(* IEC 61131-3 sources: LAxisCtrl/src/blocks (part 2) *)

                            // Write MC_Command outputs to internal variable
                            _exeOfBasicMotion := 16#0;
                            _exeOfBasicMotion.%X0 := _instHalt.Busy;
                            _exeOfBasicMotion.%X1 := _instHalt.Done;
                            _exeOfBasicMotion.%X2 := _instHalt.CommandAborted;
                            _exeOfBasicMotion.%X3 := _instHalt.Error;

                        JOG_FORWARD_SELECTED, JOG_BACKWARD_SELECTED, JOG_FW_AND_BW_SELECTED:
                            // Additional features (applicative): Jog mode incremental

                            CASE _jogMode OF
                                JOG_MODE_CONTINUOUS:

                                    // No additional feature
                                    // Firstcycle of command
                                    IF (_firstCycleBasicMotion = TRUE) THEN
                                        // Copy no dynamics into static variables because changes are accepted by MC_MoveJog immediately (enable)
                                        _instMoveJog(Axis := _refSpeedAxis^,
                                                     JogForward := FALSE,
                                                     JogBackward := FALSE);
                                    END_IF;

                                    // Call MC_Command
                                    _instMoveJog(Axis := _refSpeedAxis^,
                                                 JogForward := _basicCommand.%X2,
                                                 JogBackward := _basicCommand.%X3,
                                                 Velocity := config.jog.velocity,
                                                 Acceleration := config.jog.acceleration,
                                                 Deceleration := config.jog.deceleration,
                                                 PositionControlled := config.jog.positionControlled,
                                                 Jerk := config.jog.jerk);

                                    // Evaluate MC_Command
                                    IF (_instMoveJog.Busy = FALSE) AND
                                        (_instMoveJog.Error = FALSE) AND
                                        (_instMoveJog.CommandAborted = FALSE) AND
                                        (_instMoveJog.InVelocity = FALSE)
                                    THEN
                                        // Return to NO_SELECTION if command finished
                                        _basicMotionState := NO_SELECTION;

                                    ELSIF (_instMoveJog.Error = TRUE) THEN
                                        // Errorhandling
                                        _status := AxisStatus#ERR_MC_MOVEJOG;
                                        _statusText := STRING#'ERR_MC_MOVEJOG';
                                        _errorAutoCleared := TRUE;
                                        _diagnostics.subfunctionStatus := _instMoveJog.ErrorId;
                                        _subfunctionStatus := _instMoveJog.ErrorId;
                                        // Set next state
                                        _basicMotionState := NO_SELECTION;
                                        _state := AXIS_STOP_ON_ERROR_SELECTION;
                                        // ELSE
                                        //   ; // Command selected
                                    END_IF;

                                    // Write MC_Command outputs to internal variable
                                    _exeOfBasicMotion := 16#0;
                                    _exeOfBasicMotion.%X0 := _instMoveJog.Busy;
                                    _exeOfBasicMotion.%X2 := _instMoveJog.CommandAborted;
                                    _exeOfBasicMotion.%X3 := _instMoveJog.Error;
                                    _exeOfBasicMotion.%X4 := _instMoveJog.InVelocity;

                                JOG_MODE_CONTINUE_INCREMENT, JOG_MODE_NEW_INCREMENT:

                                    // This case is additional feature (MC_MOVERELATIVE and MC_HALT internal used)
                                    CASE _exeOfBasicMotion OF
                                        CMD_BUSY:
                                            // Firstcycle of command
                                            IF (_firstCycleBasicMotion = TRUE) THEN // New rising edge at JogForward or JogBackward
                                                // Check for only one Jog direction selected (Forward OR Backward)
                                                IF (_basicCommand.%X2 XOR _basicCommand.%X3) // Only one direction selected
                                                THEN
                                                    // Reset MOVERELATIVE command
                                                    _instMoveRelative(Axis := _refPosAxis^,
                                                                      Execute := FALSE);
                                                    // Reset HALT command
                                                    _instHalt(Axis := _refSpeedAxis^,
                                                              Execute := FALSE);

                                                    // Set new Increment if direction changed necessary
                                                    IF (_resetIncJog = FALSE) THEN
                                                        IF ((_incJogDirectionOld = FORWARD_DIR) AND (_basicCommand.%X2 = TRUE)) OR
                                                            ((_incJogDirectionOld = BACKWARD_DIR) AND (_basicCommand.%X3 = TRUE))
                                                        THEN
                                                            ; // Direction of last jog process same as current --> continue Jog
                                                        ELSE
                                                            _resetIncJog := TRUE;
                                                        END_IF;
                                                    END_IF;

                                                    // Determine distance for positioning command (relative)
                                                    IF (config.jog.mode = JOG_MODE_NEW_INCREMENT) // In this mode a new increment is always set
                                                        OR ((config.jog.mode = JOG_MODE_CONTINUE_INCREMENT) AND (_resetIncJog = TRUE))
                                                    THEN
                                                        _resetIncJog := FALSE;
                                                        // New increment
                                                        IF (_refPosAxis <> NULL) THEN // Axis type is TO_PositioningAxis or TO_SynchronousAxis
                                                            _incJogStartPosition := _refPosAxis^.Position;
                                                        ELSE // Invalid TO specification
                                                            _incJogStartPosition := 0.0;
                                                        END_IF;
                                                        _increment := Abs(config.jog.increment); // absolute Distance for increment
                                                        IF (_basicCommand.%X2 = TRUE) THEN
                                                            // JogForward selected
                                                            _position := Abs(config.jog.increment);
                                                            _increment := _position;
                                                            _incJogDirectionOld := FORWARD_DIR;
                                                        ELSIF (_basicCommand.%X3 = TRUE) THEN
                                                            // JogBackward selected
                                                            _position := -Abs(config.jog.increment);
                                                            _increment := _position;
                                                            _incJogDirectionOld := BACKWARD_DIR;
                                                        ELSE
                                                            // Normal not possible to reach ELSE-branch
                                                            _incJogDirectionOld := 0;
                                                        END_IF;
                                                    ELSE
                                                        // Check for modulo axis
                                                        IF (_refPosAxis <> NULL) THEN // Axis type is TO_PositioningAxis or TO_SynchronousAxis
                                                            tempBool := _refPosAxis^.Modulo.Enable;
                                                        ELSE // Invalid TO specification
                                                            tempBool := FALSE;
                                                        END_IF;

                                                        IF (tempBool = FALSE) THEN
                                                            // No Modulo enabled
                                                            // Continue increment
                                                            IF (_refPosAxis <> NULL) THEN // Axis type is TO_PositioningAxis or TO_SynchronousAxis
                                                                tempLReal := _refPosAxis^.Position;
                                                            ELSE // Invalid TO specification
                                                                tempLReal := 0.0;
                                                            END_IF;

                                                            _position := (_incJogStartPosition + _increment) - tempLReal;
                                                            // Distance := setpoint - actualvalue
                                                        ELSE
                                                            // Modulo enabled
                                                            _position := _incJogDistance;
                                                        END_IF;
                                                    END_IF;
                                                    _incJogSubState := INC_JOG_START;

                                                    // Store Dynamics
                                                    _basicVelocity := Abs(config.jog.velocity);
                                                    _basicAcceleration := config.jog.acceleration;
                                                    _basicDeceleration := config.jog.deceleration;
                                                    _basicJerk := config.jog.jerk;
                                                ELSE
                                                    // Errorhandling - Invalid direction (forward and backward selected)
                                                    _status := AxisStatus#ERR_INVALID_JOG_DIR;
                                                    _statusText := STRING#'ERR_INVALID_JOG_DIR';
                                                    _errorAutoCleared := TRUE;
                                                    _diagnostics.subfunctionStatus := WORD#0000;
                                                    _subfunctionStatus := AxisStatus#STATUS_NO_CALL;
                                                    _diagnostics.basicMotionState := _basicMotionState;
                                                    // Set next state
                                                    _state := AXIS_STOP_ON_ERROR_SELECTION;
                                                    _basicMotionState := NO_SELECTION;
                                                    _exeOfBasicMotion := CMD_ERROR;
                                                    _incJogSubState := INC_JOG_IDLE;
                                                END_IF;

                                            ELSIF ((_basicCommand.%X2 = FALSE) AND (_basicCommand.%X3 = FALSE)) // No jog input selected --> Stop moving
                                                AND (_incJogSubState <> INC_JOG_STOP)
                                            THEN
                                                // Reset HALT command
                                                _instHalt(Axis := _refSpeedAxis^,
                                                          Execute := FALSE);
                                                _incJogSubState := INC_JOG_STOP;
                                                IF (_refPosAxis <> NULL) THEN // Axis type is TO_PositioningAxis or TO_SynchronousAxis
                                                    _incJogDistance := _refPosAxis^.StatusPositioning.Distance;
                                                ELSE // Invalid TO specification
                                                    _incJogDistance := 0.0;
                                                END_IF;

                                            ELSIF (_basicCommand.%X2 = TRUE) AND (_basicCommand.%X3 = TRUE) // jogForward and jogBackward selected - Error
                                            THEN
                                                // Reset HALT command
                                                _instHalt(Axis := _refSpeedAxis^,
                                                         Execute := FALSE);
                                                _incJogSubState := INC_JOG_STOP;
                                                // Errorhandling
                                                _status := AxisStatus#ERR_INVALID_JOG_DIR;
                                                _statusText := STRING#'ERR_INVALID_JOG_DIR';
                                                _errorAutoCleared := TRUE;
                                                _diagnostics.subfunctionStatus := WORD#0000;
                                                _subfunctionStatus := AxisStatus#STATUS_NO_CALL;
                                                // Set next state
                                                _exeOfBasicMotion := CMD_ERROR;
                                                _basicMotionState := NO_SELECTION;
                                                _state := AXIS_STOP_ON_ERROR_SELECTION;
                                            // ELSE
                                                //   ; // Command running
                                            END_IF;

                                            // Select motion
                                            CASE _incJogSubState OF
                                                INC_JOG_IDLE:
                                                    ; // Do nothing - Error occurred (jogforward and jogbackward are set in firstCycle of operation)

                                                INC_JOG_START: // Run jog operation --> Motion stops automatically if increment complete
                                                    _instMoveRelative(Axis := _refPosAxis^,
                                                                    Execute := TRUE,
                                                                    Distance := _position,
                                                                    Velocity := _basicVelocity,
                                                                    Acceleration := _basicAcceleration,
                                                                    Deceleration := _basicDeceleration,
                                                                    Jerk := _basicJerk);

                                                // Evaluate MC_Command
                                                IF (_instMoveRelative.Done = TRUE) THEN
                                                    // Increment completed
                                                    _resetIncJog := TRUE;
                                                    // Set next state
                                                    _exeOfBasicMotion := CMD_DONE;
                                                    _incJogSubState := INC_JOG_IDLE;

                                                ELSIF (_instMoveRelative.Error = TRUE) THEN
                                                    _resetIncJog := TRUE;
                                                    // Errorhandling
                                                    _status := AxisStatus#ERR_MC_MOVERELATIVE;
                                                    _statusText := STRING#'ERR_MC_MOVERELATIVE';
                                                    _errorAutoCleared := TRUE;
                                                    _diagnostics.subfunctionStatus := _instMoveRelative.ErrorId;
                                                    _subfunctionStatus := _instMoveRelative.ErrorId;
                                                    // Set next state
                                                    _state := AXIS_STOP_ON_ERROR_SELECTION;
                                                    _basicMotionState := NO_SELECTION;
                                                    _exeOfBasicMotion := CMD_ERROR;
                                                    _incJogSubState := INC_JOG_IDLE;

                                                ELSIF (_instMoveRelative.CommandAborted = TRUE) THEN
                                                    _resetIncJog := TRUE;
                                                    _exeOfBasicMotion := CMD_ABORTED;
                                                    _incJogSubState := INC_JOG_IDLE;
                                                    // ELSE
                                                    //   ; // Wait for next state
                                                END_IF;

                                                INC_JOG_STOP: // Executed if inputs are reset --> Stop jog operation OR if jogForward and jogBackward are set --> Error and stop axis
                                                    _instHalt(Axis := _refSpeedAxis^,
                                                              Execute := TRUE,
                                                              Deceleration := _basicDeceleration,
                                                              AbortAcceleration := FALSE,
                                                              Jerk := _basicJerk,
                                                              Mode := 0); // Mode := 0 "The basic motion and the superimposed motion are stopped." MC_Halt instance is also used for input 'stop', where the 'haltMode' can now be specified via config

                                                    // Evaluate MC_Command
                                                    IF (_instHalt.Done = TRUE) THEN
                                                        // Set next state
                                                        _exeOfBasicMotion := CMD_END_PROCESS;
                                                        _incJogSubState := INC_JOG_IDLE;

                                                    ELSIF (_instHalt.Error = TRUE) THEN
                                                        _resetIncJog := TRUE;
                                                        // Errorhandling
                                                        _status := AxisStatus#ERR_MC_HALT;
                                                        _statusText := STRING#'ERR_MC_HALT';
                                                        _errorAutoCleared := TRUE;
                                                        _diagnostics.subfunctionStatus := _instHalt.ErrorId;
                                                        _subfunctionStatus := _instHalt.ErrorId;
                                                        // Set next state
                                                        _state := AXIS_STOP_ON_ERROR_SELECTION;
                                                        _basicMotionState := NO_SELECTION;
                                                        _exeOfBasicMotion := CMD_ERROR;
                                                        _incJogSubState := INC_JOG_IDLE;

                                                    ELSIF (_instHalt.CommandAborted = TRUE) THEN
                                                        _resetIncJog := TRUE;
                                                        // Set next state
                                                        _incJogSubState := INC_JOG_IDLE;
                                                        _exeOfBasicMotion := CMD_ABORTED;
                                                    // ELSE
                                                        //   ; // Wait for stopping axis
                                                    END_IF;
                                                ELSE
                                                    // Errorhandling
                                                    _status := AxisStatus#ERR_UNDEFINED_INCREMENTAL_JOG_SUBSTATE;
                                                    _statusText := STRING#'ERR_UNDEFINED_INCREMENTAL_JOG_SUBSTATE';
                                                    _errorUserCleared := TRUE;
                                                    _diagnostics.subfunctionStatus := WORD#0000;
                                                    _subfunctionStatus := AxisStatus#STATUS_NO_CALL;
                                                    // Set errorstate
                                                    _state := FB_ERROR;
                                                END_CASE;

                                        CMD_DONE,
                                        CMD_ABORTED,
                                        CMD_ERROR,
                                        CMD_END_PROCESS:
                                            // Return to NO_SELECTION if command finished
                                            IF (_basicCommand.%X2 = FALSE) AND (_basicCommand.%X3 = FALSE) THEN
                                                // jogForward and jogbackward inputs are reset
                                                _exeOfBasicMotion := CMD_BUSY;
                                                _basicMotionState := NO_SELECTION;
                                            // ELSE
                                                //   ; // Wait for falling edge at inputs for jog
                                            END_IF;
                                    ELSE
                                        // Errorhandling
                                        _status := AxisStatus#ERR_UNDEFINED_INCREMENTAL_JOG_STATE;
                                        _statusText := STRING#'ERR_UNDEFINED_INCREMENTAL_JOG_STATE';
                                        _errorUserCleared := TRUE;
                                        _diagnostics.subfunctionStatus := WORD#0000;
                                        _subfunctionStatus := AxisStatus#STATUS_NO_CALL;
                                        _diagnostics.basicMotionState := _basicMotionState;
                                        // Set errorstate
                                        _state := FB_ERROR;
                                    END_CASE;

                            ELSE
                                // Errorhandling - Invalid jog state
                                _status := AxisStatus#ERR_INVALID_JOG_MODE;
                                _statusText := STRING#'#ERR_INVALID_JOG_MODE';
                                _errorAutoCleared := TRUE;
                                _diagnostics.subfunctionStatus := WORD#0000;
                                _subfunctionStatus := AxisStatus#STATUS_NO_CALL;
                                // Set next state
                                _state := AXIS_STOP_ON_ERROR_SELECTION;
                                _basicMotionState := NO_SELECTION;
                            END_CASE;

                        MOVE_VELOCITY_SELECTED:
                            // Additional features (applicative): Change setpoint on the fly (Velocity)

                            // Firstcycle of command
                            IF (_firstCycleBasicMotion = TRUE) THEN
                                // Reset MC_MOVEVELOCITY command
                                _instMoveVelocity(Axis := _refSpeedAxis^,
                                                    Execute := FALSE);

                                _velocityChangeOnTheFly := config.moveVelocity.velocityChangeOnTheFly;

                                _instMoveVelocity.Velocity := config.moveVelocity.velocity;
                                _basicVelocity := config.moveVelocity.velocity;

                                _instMoveVelocity.Acceleration := config.moveVelocity.acceleration;
                                _instMoveVelocity.Deceleration := config.moveVelocity.deceleration;
                                _instMoveVelocity.Jerk := config.moveVelocity.jerk;
                                _instMoveVelocity.Direction := config.moveVelocity.direction;
                                _instMoveVelocity.PositionControlled := config.moveVelocity.positionControlled;
                                _instMoveVelocity.Current := FALSE;

                            ELSIF (_velocityChangeOnTheFly = TRUE) AND (config.moveVelocity.velocity <> _basicVelocity) // Velocity changed
                                AND (_instMoveVelocity.CommandAborted = FALSE)
                            THEN
                                // Reset MC_MOVEVELOCITY command
                                _instMoveVelocity(Axis := _refSpeedAxis^,
                                                Execute := FALSE);

                                _instMoveVelocity.Velocity := config.moveVelocity.velocity;
                                _basicVelocity := config.moveVelocity.velocity;

                                // Copy also dynamics
                                _instMoveVelocity.Acceleration := config.moveVelocity.acceleration;
                                _instMoveVelocity.Deceleration := config.moveVelocity.deceleration;
                                _instMoveVelocity.Jerk := config.moveVelocity.jerk;
                                _instMoveVelocity.Direction := config.moveVelocity.direction;
                                _instMoveVelocity.PositionControlled := config.moveVelocity.positionControlled;
                            END_IF;

                            // Call MC_Command
                            _instMoveVelocity(Axis := _refSpeedAxis^,
                                              Execute := _basicCommand.%X4 OR _firstCycleBasicMotion); // Input: moveVelocity

                            // Evaluate MC_Command
                            IF (_instMoveVelocity.Busy = FALSE) AND
                                (_instMoveVelocity.Error = FALSE) AND
                                (_instMoveVelocity.CommandAborted = FALSE) AND
                                (_instMoveVelocity.InVelocity = FALSE)
                            THEN
                                // Return to NO_SELECTION if command finished
                                _basicMotionState := NO_SELECTION;

                            ELSIF (_instMoveVelocity.Error = TRUE) THEN
                                // Errorhandling
                                _status := AxisStatus#ERR_MC_MOVEVELOCITY;
                                _statusText := STRING#'ERR_MC_MOVEVELOCITY';
                                _errorAutoCleared := TRUE;
                                _diagnostics.subfunctionStatus := _instMoveVelocity.ErrorId;
                                _subfunctionStatus := _instMoveVelocity.ErrorId;
                                _velocityChangeOnTheFly := FALSE;
                                // Set next state
                                _state := AXIS_STOP_ON_ERROR_SELECTION;
                                _basicMotionState := NO_SELECTION;
                                // ELSE
                                //   ; // Command selected
                            END_IF;

                            // Write MC_Command outputs to internal variable
                            _exeOfBasicMotion := 16#0;
                            _exeOfBasicMotion.%X0 := _instMoveVelocity.Busy;
                            _exeOfBasicMotion.%X2 := _instMoveVelocity.CommandAborted;
                            _exeOfBasicMotion.%X3 := _instMoveVelocity.Error;
                            _exeOfBasicMotion.%X4 := _instMoveVelocity.InVelocity;

                        POS_RELATIVE_SELECTED:
                            // Additional features (applicative): Specified direction

                            // Firstcycle of command
                            IF (_firstCycleBasicMotion = TRUE) THEN
                                // Configurate the direction of rotation
                                IF ((config.posRelative.direction = 0) AND (config.posRelative.distance >= 0.0)) // Sign of distance is evaluated
                                    OR (config.posRelative.direction = FORWARD_DIR) // Forward direction
                                THEN
                                    _position := Abs(config.posRelative.distance);
                                    // Reset MC_MOVERELATIVE command
                                    _instMoveRelative(Axis := _refPosAxis^,
                                                      Execute := FALSE,
                                                      Distance := _position,
                                                      Velocity := config.posRelative.velocity,
                                                      Acceleration := config.posRelative.acceleration,
                                                      Deceleration := config.posRelative.deceleration,
                                                      Jerk := config.posRelative.jerk);
                                    _applicativeBasicMotionError := FALSE;

                                ELSIF ((config.posRelative.direction = 0) AND (config.posRelative.distance < 0.0)) // Sign of distance is evaluated
                                    OR (config.posRelative.direction = BACKWARD_DIR) // Backward direction
                                THEN
                                    _position := -Abs(config.posRelative.distance);
                                    // Reset MC_MOVERELATIVE command
                                    _instMoveRelative(Axis := _refPosAxis^,
                                                      Execute := FALSE,
                                                      Distance := _position,
                                                      Velocity := config.posRelative.velocity,
                                                      Acceleration := config.posRelative.acceleration,
                                                      Deceleration := config.posRelative.deceleration,
                                                      Jerk := config.posRelative.jerk);

                                    _applicativeBasicMotionError := FALSE;
                                ELSE
                                    // Errorhandling - Invalid direction
                                    _status := AxisStatus#ERR_INVALID_POS_RELATIVE_DIR;
                                    _statusText := STRING#'ERR_INVALID_POS_RELATIVE_DIR';
                                    _errorAutoCleared := TRUE;
                                    _diagnostics.subfunctionStatus := WORD#0000;
                                    _subfunctionStatus := AxisStatus#STATUS_NO_CALL;
                                    _applicativeBasicMotionError := TRUE;
                                    // Set next state
                                    _state := AXIS_STOP_ON_ERROR_SELECTION;
                                    _basicMotionState := NO_SELECTION;
                                END_IF;
                            END_IF;

                            IF (_applicativeBasicMotionError = FALSE) THEN
                                // Call MC_Command
                                _instMoveRelative(Axis := _refPosAxis^,
                                                  Execute := _basicCommand.%X5 OR _firstCycleBasicMotion); // Input: posRelative

                                // Evaluate MC_Command
                                IF (_instMoveRelative.Busy = FALSE) AND
                                    (_instMoveRelative.Error = FALSE) AND
                                    (_instMoveRelative.Done = FALSE) AND
                                    (_instMoveRelative.CommandAborted = FALSE)
                                THEN
                                    // Return to NO_SELECTION if command finished
                                    _basicMotionState := NO_SELECTION;

                                ELSIF (_instMoveRelative.Error = TRUE) THEN
                                    // Errorhandling
                                    _status := AxisStatus#ERR_MC_MOVERELATIVE;
                                    _statusText := STRING#'ERR_MC_MOVERELATIVE';
                                    _errorAutoCleared := TRUE;
                                    _diagnostics.subfunctionStatus := _instMoveRelative.ErrorId;
                                    _subfunctionStatus := _instMoveRelative.ErrorId;
                                    // Set next state
                                    _state := AXIS_STOP_ON_ERROR_SELECTION;
                                    _basicMotionState := NO_SELECTION;
                                // ELSE
                                    //   ; // Command selected
                                END_IF;

                                // Write MC_Command outputs to internal variable
                                _exeOfBasicMotion := 16#0;
                                _exeOfBasicMotion.%X0 := _instMoveRelative.Busy;
                                _exeOfBasicMotion.%X1 := _instMoveRelative.Done;
                                _exeOfBasicMotion.%X2 := _instMoveRelative.CommandAborted;
                                _exeOfBasicMotion.%X3 := _instMoveRelative.Error;
                            // ELSE
                                //   ; // Direction not valid
                            END_IF;

                        POS_ABSOLUTE_SELECTED:
                            // Additional features (applicative): Change setpoint on the fly (Velocity and Position)

                            // Firstcycle of command
                            IF (_firstCycleBasicMotion = TRUE) THEN
                                // Reset MC_MOVEABSOLUTE command
                                _instMoveAbsolute(Axis := _refPosAxis^,
                                                  Execute := FALSE);

                                _instMoveAbsolute.Position := config.posAbsolute.position;
                                _position := config.posAbsolute.position;
                                _instMoveAbsolute.Velocity := config.posAbsolute.velocity;
                                _basicVelocity := config.posAbsolute.velocity;

                                _instMoveAbsolute.Acceleration := config.posAbsolute.acceleration;
                                _instMoveAbsolute.Deceleration := config.posAbsolute.deceleration;
                                _instMoveAbsolute.Jerk := config.posAbsolute.jerk;
                                _instMoveAbsolute.Direction := config.posAbsolute.direction;

                                _velocityChangeOnTheFly := config.posAbsolute.velocityChangeOnTheFly;
                                _positionChangeOnTheFly := config.posAbsolute.positionChangeOnTheFly;

                            ELSIF (((_velocityChangeOnTheFly = TRUE) AND (config.posAbsolute.velocity <> _basicVelocity))
                                OR ((_positionChangeOnTheFly = TRUE) AND (config.posAbsolute.position <> _position)))
                                AND (_instMoveAbsolute.CommandAborted = FALSE)
                            THEN
                                // Reset MC_MOVEABSOLUTE command
                                _instMoveAbsolute(Axis := _refPosAxis^,
                                                  Execute := FALSE);

                                IF (_velocityChangeOnTheFly = TRUE) THEN // Apply the new velocity value
                                    _instMoveAbsolute.Velocity := config.posAbsolute.velocity;
                                    _basicVelocity := config.posAbsolute.velocity;

                                    // Copy also dynamics
                                    _instMoveAbsolute.Acceleration := config.posAbsolute.acceleration;
                                    _instMoveAbsolute.Deceleration := config.posAbsolute.deceleration;
                                    _instMoveAbsolute.Jerk := config.posAbsolute.jerk;
                                    _instMoveAbsolute.Direction := config.posAbsolute.direction;
                                END_IF;

                                IF (_positionChangeOnTheFly = TRUE) THEN // Apply the new position value
                                    _instMoveAbsolute.Position := config.posAbsolute.position;
                                    _position := config.posAbsolute.position;

                                    // Copy also dynamics
                                    _instMoveAbsolute.Velocity := config.posAbsolute.velocity;
                                    _instMoveAbsolute.Acceleration := config.posAbsolute.acceleration;
                                    _instMoveAbsolute.Deceleration := config.posAbsolute.deceleration;
                                    _instMoveAbsolute.Jerk := config.posAbsolute.jerk;
                                    _instMoveAbsolute.Direction := config.posAbsolute.direction;
                                END_IF;
                            END_IF;

                            _instMoveAbsolute(Axis := _refPosAxis^,
                                              Execute := _basicCommand.%X6 OR _firstCycleBasicMotion); // Input: posAbsolute

                            // Evaluate MC_Command
                            IF (_instMoveAbsolute.Busy = FALSE) AND
                                (_instMoveAbsolute.Error = FALSE) AND
                                (_instMoveAbsolute.Done = FALSE) AND
                                (_instMoveAbsolute.CommandAborted = FALSE)
                            THEN
                                // Return to NO_SELECTION if command finished
                                _basicMotionState := NO_SELECTION;

                            ELSIF (_instMoveAbsolute.Error = TRUE) THEN
                                // Errorhandling
                                _status := AxisStatus#ERR_MC_MOVEABSOLUTE;
                                _statusText := STRING#'ERR_MC_MOVEABSOLUTE';
                                _errorAutoCleared := TRUE;
                                _diagnostics.subfunctionStatus := _instMoveAbsolute.ErrorId;
                                _subfunctionStatus := _instMoveAbsolute.ErrorId;
                                _velocityChangeOnTheFly := FALSE;
                                _positionChangeOnTheFly := FALSE;
                                // Set next state
                                _state := AXIS_STOP_ON_ERROR_SELECTION;
                                _basicMotionState := NO_SELECTION;
                            END_IF;

                            // Write MC_Command outputs to internal variable
                            _exeOfBasicMotion := 16#0;
                            _exeOfBasicMotion.%X0 := _instMoveAbsolute.Busy;
                            _exeOfBasicMotion.%X1 := _instMoveAbsolute.Done;
                            _exeOfBasicMotion.%X2 := _instMoveAbsolute.CommandAborted;
                            _exeOfBasicMotion.%X3 := _instMoveAbsolute.Error;

                        ACTIVE_HOMING_SELECTED:
                            // Additional feature (applicative): homing on fixed stop

                            // Firstcycle of command
                            IF (_firstCycleBasicMotion = TRUE) THEN
                                _activeHomingState := config.homing.extendedMode;
                                _exeOfBasicMotion := CMD_BUSY;
                                _passiveHomingState := NO_HOMING_ACTIVE;
                            END_IF;

                            // Selection of extended homing mode
                            CASE _activeHomingState OF
                                STANDARD_HOMING:
                                    // No additional features

                                    // Firstcycle of command
                                    IF (_firstCycleBasicMotion = TRUE) THEN
                                        // Reset MC_HOME command
                                        _instHome(Axis := _refAxis^,
                                                  Execute := FALSE,
                                                  Position := config.homing.position,
                                                  Mode := config.homing.mode,
                                                  Sensor := config.homing.sensor);
                                    END_IF;

                                    // Call MC_Command

                                    _instHome(Axis := _refAxis^,
                                              Execute := _basicCommand.%X10 OR _firstCycleBasicMotion); // Input: homing

                                    // Evaluate MC_Command
                                    IF (_instHome.Busy = FALSE) AND
                                        (_instHome.Done = FALSE) AND
                                        (_instHome.CommandAborted = FALSE) AND
                                        (_instHome.Error = FALSE)
                                    THEN
                                        // Return to NO_SELECTION if command finished
                                        _activeHomingState := STANDARD_HOMING;
                                        _basicMotionState := NO_SELECTION;

                                    ELSIF (_instHome.Error = TRUE) THEN
                                        // Errorhandling
                                        _status := AxisStatus#ERR_MC_HOME;
                                        _statusText := STRING#'ERR_MC_HOME';
                                        _errorAutoCleared := TRUE;
                                        _diagnostics.subfunctionStatus := _instHome.ErrorId;
                                        _subfunctionStatus := _instHome.ErrorId;
                                        _state := AXIS_STOP_ON_ERROR_SELECTION;
                                        _basicMotionState := NO_SELECTION;
                                        // ELSE
                                        //   ; // Command selected
                                    END_IF;

                                    _exeOfBasicMotion := 16#0;
                                    _exeOfBasicMotion.%X0 := _instHome.Busy;
                                    _exeOfBasicMotion.%X1 := _instHome.Done;
                                    _exeOfBasicMotion.%X2 := _instHome.CommandAborted;
                                    _exeOfBasicMotion.%X3 := _instHome.Error;

                                HOMING_ON_FIXED_STOP,
                                HOMING_ON_FIXED_STOP_WITH_MOVING_OUT_OF_CLAMPING,
                                HOMING_ON_FIXED_STOP_WITH_MOVING_TO_TARGET_POSITION:
                                    // This case is additional feature (MC_MOVEVELOCITY and MC_HOME internal used)

                                    CASE _exeOfBasicMotion OF
                                        CMD_BUSY:
                                            // Firstcycle of command
                                            IF (_firstCycleBasicMotion = TRUE) THEN

                                                // Read operative sensor
                                                IF (_refPosAxis <> NULL) THEN // Axis type is TO_PositioningAxis or TO_SynchronousAxis
                                                    tempIndex := TO_INT(_refPosAxis^.OperativeSensor);
                                                ELSE // Invalid TO specification
                                                    tempIndex := 1;
                                                END_IF;

                                                IF (tempIndex < 1) THEN
                                                    tempIndex := 1;
                                                END_IF;

                                                IF (_refPosAxis <> NULL) THEN // Axis type is TO_PositioningAxis or TO_SynchronousAxis
                                                    tempDInt := _refPosAxis^.Sensor[tempIndex].ActiveHoming.Direction;
                                                ELSE // Invalid TO specification
                                                    tempDInt := 0; // Positive direction
                                                END_IF;

                                                IF (tempDInt = 0)
                                                THEN
                                                    // Positive direction
                                                    _direction := FORWARD_DIR;
                                                ELSE
                                                    // Negative direction
                                                    _direction := BACKWARD_DIR;
                                                END_IF;

                                                // Check if homing on fixed stop is allowed

                                                IF (_refPosAxis <> NULL) THEN // Axis type is TO_PositioningAxis or TO_SynchronousAxis
                                                    tempBool := _refPosAxis^.Modulo.Enable;
                                                    tempLReal := _refPosAxis^.Homing.ReferencingVelocity;
                                                ELSE // Invalid TO specification
                                                    tempBool := FALSE;
                                                    tempLReal := 0.0;
                                                END_IF;

                                                IF (tempBool = TRUE) THEN
                                                    // Modulo enabled - Errorhandling
                                                    _status := AxisStatus#ERR_MODULO_NOT_ALLOWED;
                                                    _statusText := STRING#'ERR_MODULO_NOT_ALLOWED';
                                                    _errorAutoCleared := TRUE;
                                                    _diagnostics.subfunctionStatus := WORD#0000;
                                                    _subfunctionStatus := AxisStatus#STATUS_NO_CALL;
                                                    _diagnostics.basicMotionState := _basicMotionState;
                                                    // Set next state
                                                    _state := AXIS_STOP_ON_ERROR_SELECTION;
                                                    _basicMotionState := NO_SELECTION;
                                                    _activeHomingState := STANDARD_HOMING;
                                                    _homingSubState := HOMING_IDLE;

                                                ELSIF (config.homing.extendedModeTorqueLimit = 0.0) // Torque limit 0.0 in config
                                                THEN
                                                    // Errorhandling -  Torque value 0.0 configured
                                                    _status := AxisStatus#ERR_INVALID_TORQUE_LIMIT;
                                                    _statusText := STRING#'ERR_INVALID_TORQUE_LIMIT';
                                                    _errorAutoCleared := TRUE;
                                                    _diagnostics.subfunctionStatus := WORD#0000;
                                                    _subfunctionStatus := AxisStatus#STATUS_NO_CALL;
                                                    _diagnostics.basicMotionState := _basicMotionState;
                                                    // Set next state
                                                    _state := AXIS_STOP_ON_ERROR_SELECTION;
                                                    _basicMotionState := NO_SELECTION;
                                                    _activeHomingState := STANDARD_HOMING;
                                                    _homingSubState := HOMING_IDLE;

                                                ELSIF (tempLReal = 0.0)
                                                THEN
                                                    // Errorhandling -  Velocity 0 configured
                                                    _status := AxisStatus#ERR_INVALID_VELOCITY;
                                                    _statusText := STRING#'ERR_INVALID_VELOCITY';
                                                    _errorAutoCleared := TRUE;
                                                    _diagnostics.subfunctionStatus := WORD#0000;
                                                    _subfunctionStatus := AxisStatus#STATUS_NO_CALL;
                                                    _diagnostics.basicMotionState := _basicMotionState;
                                                    // Set next state
                                                    _state := AXIS_STOP_ON_ERROR_SELECTION;
                                                    _basicMotionState := NO_SELECTION;
                                                    _activeHomingState := STANDARD_HOMING;
                                                    _homingSubState := HOMING_IDLE;

                                                ELSIF (_activeHomingState = HOMING_ON_FIXED_STOP_WITH_MOVING_TO_TARGET_POSITION) // condition modified (check target pos. only if extendedMode = 2)
                                                    AND
                                                    ((config.homing.extendedModeTargetPosition > config.homing.position) AND (_direction = FORWARD_DIR)
                                                    OR (config.homing.extendedModeTargetPosition < config.homing.position) AND (_direction = BACKWARD_DIR))
                                                THEN
                                                    // Errorhandling -  Invalid target position for extended homing mode "2: Homing on fixed stop with moving to target position"
                                                    _status := AxisStatus#ERR_INVALID_TARGET_POSITION;
                                                    _statusText := STRING#'ERR_INVALID_TARGET_POSITION';
                                                    _errorAutoCleared := TRUE;
                                                    _diagnostics.subfunctionStatus := WORD#0000;
                                                    _subfunctionStatus := AxisStatus#STATUS_NO_CALL;
                                                    _diagnostics.basicMotionState := _basicMotionState;
                                                    // Set next state
                                                    _state := AXIS_STOP_ON_ERROR_SELECTION;
                                                    _basicMotionState := NO_SELECTION;
                                                    _activeHomingState := STANDARD_HOMING;
                                                    _homingSubState := HOMING_IDLE;

                                                ELSE
                                                    // Store dynamic values
                                                    _homingPosition := config.homing.position;
                                                    _basicVelocity := tempLReal;
                                                    IF (_refPosAxis <> NULL) THEN // Axis type is TO_PositioningAxis or TO_SynchronousAxis
                                                        _basicAcceleration := _refPosAxis^.DynamicDefaults.Acceleration;
                                                        _basicDeceleration := _refPosAxis^.DynamicDefaults.Deceleration;
                                                        _basicJerk := _refPosAxis^.DynamicDefaults.Jerk;
                                                    ELSE // Invalid TO specification
                                                        _basicAcceleration := -1.0;
                                                        _basicDeceleration := -1.0;
                                                        _basicJerk := 0.0; // No Jerk
                                                    END_IF;

                                                    _torqueLimitingState := FIXED_STOP_DETECTION_ACTIVE;
                                                    // Reset MC_Commands
                                                    _instHome(Axis := _refAxis^,
                                                              Execute := FALSE,
                                                              Position := _homingPosition,
                                                              //  Mode := statHomingMode,
                                                              Sensor := 0);

                                                    _instMoveVelocity(Axis := _refSpeedAxis^,
                                                                      Execute := FALSE,
                                                                      Velocity := _basicVelocity,
                                                                      Acceleration := _basicAcceleration,
                                                                      Deceleration := _basicDeceleration,
                                                                      Jerk := _basicJerk,
                                                                      PositionControlled := TRUE,
                                                                      Direction := _direction);

                                                    _instMoveAbsolute(Axis := _refPosAxis^,
                                                                      Execute := FALSE,
                                                                      Velocity := Abs(_basicVelocity),
                                                                      Acceleration := _basicAcceleration,
                                                                      Deceleration := _basicDeceleration,
                                                                      Jerk := _basicJerk);

                                                    // Determine the encoder type
                                                    IF (_refPosAxis <> NULL) THEN // Axis type is TO_PositioningAxis or TO_SynchronousAxis
                                                        tempDInt := _refPosAxis^.Sensor[tempIndex]._Type;
                                                    ELSE // Invalid TO specification
                                                        tempDInt := 0; // Incremental
                                                    END_IF;

                                                    IF (tempDInt = INCREMENTAL_ENCODER) THEN
                                                        _instHome.Mode := DIRECT_HOMING; // Direct homing (absolute)
                                                    ELSE
                                                        _instHome.Mode := ABSOLUTE_ENCODER_ADJUSTMENT;
                                                    END_IF;
                                                    // Use always direct homing
                                                    //#statHomingMode := DIRECT_HOMING; // Direct homing (absolute)
                                                    // Set next state
                                                    _homingSubState := HOMING_FIXED_STOP_DETECTION;
                                                END_IF;
                                            END_IF;

                                            // Call of subStateMachine
                                            REPEAT
                                                CASE _homingSubState OF
                                                    HOMING_IDLE:
                                                        tempStateChangeActive := FALSE;
                                                        // Do nothing, no execution of homing if error occurred in first cycle

                                                    HOMING_FIXED_STOP_DETECTION:
                                                        tempStateChangeActive := FALSE;

                                                        // Start axis to detect fixed stop
                                                        _instMoveVelocity(Axis := _refSpeedAxis^,
                                                                        Execute := TRUE);

                                                        // Evaluate MC_Command
                                                        IF (tempStatusWord.%X30 = TRUE) THEN // inClamping = TRUE
                                                            // Fixed stop detected --> start homing process
                                                            _homingSubState := HOMING_PROCESS;
                                                            tempStateChangeActive := TRUE;

                                                        ELSIF (_instMoveVelocity.Error = TRUE) THEN
                                                            // Errorhandling
                                                            _status := AxisStatus#ERR_MC_MOVEVELOCITY;
                                                            _statusText := STRING#'ERR_MC_MOVEVELOCITY';
                                                            _errorAutoCleared := TRUE;
                                                            _diagnostics.subfunctionStatus := _instMoveVelocity.ErrorId;
                                                            _subfunctionStatus := _instMoveVelocity.ErrorId;
                                                            // Set next state
                                                            _state := AXIS_STOP_ON_ERROR_SELECTION;
                                                            _basicMotionState := NO_SELECTION;
                                                            _activeHomingState := STANDARD_HOMING;
                                                            _exeOfBasicMotion := CMD_ERROR;
                                                            _homingSubState := HOMING_IDLE;

                                                        ELSIF (_instMoveVelocity.CommandAborted = TRUE) THEN
                                                            // Set next state
                                                            _exeOfBasicMotion := CMD_ABORTED;
                                                            _homingSubState := HOMING_IDLE;
                                                        // ELSE
                                                            //   ;// Wait for detecting fixed stop
                                                        END_IF;

                                                    HOMING_PROCESS:
                                                        tempStateChangeActive := FALSE;
                                                        // Execute MC_HOME
                                                        _instHome(Axis := _refAxis^,
                                                                Execute := TRUE);

                                                        // Evaluate MC_Command
                                                        IF (_instHome.Done = TRUE) THEN
                                                            // MC_HOME finished - Set next state
                                                            _homingSubState := HOMING_POSITION;
                                                            tempStateChangeActive := TRUE;

                                                        ELSIF (_instHome.Error = TRUE) THEN
                                                            // Errorhandling
                                                            _status := AxisStatus#ERR_MC_HOME;
                                                            _statusText := STRING#'ERR_MC_HOME';
                                                            _errorAutoCleared := TRUE;
                                                            _diagnostics.subfunctionStatus := _instHome.ErrorId;
                                                            _subfunctionStatus := _instHome.ErrorId;
                                                            // Set next state
                                                            _state := AXIS_STOP_ON_ERROR_SELECTION;
                                                            _exeOfBasicMotion := CMD_ERROR;
                                                            _homingSubState := HOMING_IDLE;

                                                        ELSIF (_instHome.CommandAborted = TRUE) THEN
                                                            // Set next state
                                                            _exeOfBasicMotion := CMD_ABORTED;
                                                            _homingSubState := HOMING_IDLE;
                                                        // ELSE
                                                            //   ;// Wait for finish homing process
                                                        END_IF;

                                                    HOMING_POSITION:
                                                        tempStateChangeActive := FALSE;
                                                        CASE _activeHomingState OF
                                                            HOMING_ON_FIXED_STOP:
                                                                // Execute moving to homeposition
                                                                _instMoveAbsolute(Axis := _refPosAxis^,
                                                                                Execute := TRUE,
                                                                                Position := _homingPosition,
                                                                                Direction := SHORTEST_WAY_DIR);

                                                                // Evaluate MC_Command
                                                                IF (_instMoveAbsolute.Done = TRUE) THEN
                                                                    // Homeposition reached - Set next state
                                                                    _exeOfBasicMotion := CMD_DONE;
                                                                    _homingSubState := HOMING_IDLE;

                                                                ELSIF (_instMoveAbsolute.Error = TRUE) THEN
                                                                    // Errorhandling
                                                                    _status := AxisStatus#ERR_MC_MOVEABSOLUTE;
                                                                    _statusText := STRING#'ERR_MC_MOVEABSOLUTE';
                                                                    _errorAutoCleared := TRUE;
                                                                    _diagnostics.subfunctionStatus := _instMoveAbsolute.ErrorId;
                                                                    _subfunctionStatus := _instMoveAbsolute.ErrorId;
                                                                    // Set next state
                                                                    _state := AXIS_STOP_ON_ERROR_SELECTION;
                                                                    _basicMotionState := CMD_BUSY;
                                                                    _activeHomingState := STANDARD_HOMING;
                                                                    _exeOfBasicMotion := CMD_ERROR;
                                                                    _homingSubState := HOMING_IDLE;

                                                                ELSIF (_instMoveAbsolute.CommandAborted = TRUE) THEN
                                                                    // Set next state
                                                                    _exeOfBasicMotion := CMD_ABORTED;
                                                                    _homingSubState := HOMING_IDLE;
                                                                // ELSE
                                                                    //   ; // Wait for reaching homeposition
                                                                END_IF;

                                                            HOMING_ON_FIXED_STOP_WITH_MOVING_OUT_OF_CLAMPING:
                                                                // Execute moving to homeposition
                                                                IF (_refPosAxis <> NULL) THEN // Axis type is TO_PositioningAxis or TO_SynchronousAxis
                                                                    tempLReal := _refPosAxis^.Clamping.PositionTolerance;
                                                                ELSE // Invalid TO specification
                                                                    tempLReal := 0.0;
                                                                END_IF;

                                                                CASE _direction OF
                                                                    FORWARD_DIR:
                                                                        _homingPosition := _homingPosition - (DISTANCE_SCALING * tempLReal);

                                                                    BACKWARD_DIR:
                                                                        _homingPosition := _homingPosition + (DISTANCE_SCALING * tempLReal);
                                                                END_CASE;

                                                                // Execute moving to homeposition
                                                                _instMoveAbsolute(Axis := _refPosAxis^,
                                                                                Execute := TRUE,
                                                                                Position := _homingPosition,
                                                                                Direction := SHORTEST_WAY_DIR);

                                                                // Evaluate MC_Command
                                                                IF (_instMoveAbsolute.Done = TRUE) AND (_instTorqueLimiting.InClamping = FALSE) THEN
                                                                    // Homeposition reached - Set next state
                                                                    _exeOfBasicMotion := CMD_DONE;
                                                                    _homingSubState := HOMING_IDLE;

                                                                ELSIF (_instMoveAbsolute.Error = TRUE) THEN
                                                                    // Errorhandling
                                                                    _status := AxisStatus#ERR_MC_MOVEABSOLUTE;
                                                                    _statusText := STRING#'ERR_MC_MOVEABSOLUTE';
                                                                    _errorAutoCleared := TRUE;
                                                                    _diagnostics.subfunctionStatus := _instMoveAbsolute.ErrorId;
                                                                    _subfunctionStatus := _instMoveAbsolute.ErrorId;
                                                                    // Set next state
                                                                    _state := AXIS_STOP_ON_ERROR_SELECTION;
                                                                    _basicMotionState := CMD_BUSY;
                                                                    _activeHomingState := STANDARD_HOMING;
                                                                    _exeOfBasicMotion := CMD_ERROR;
                                                                    _homingSubState := HOMING_IDLE;

                                                                ELSIF (_instMoveAbsolute.CommandAborted = TRUE) THEN
                                                                    // Set next state
                                                                    _exeOfBasicMotion := CMD_ABORTED;
                                                                    _homingSubState := HOMING_IDLE;

                                                                // ELSE
                                                                    //   ; // Wait for reaching homeposition
                                                                END_IF;

                                                            HOMING_ON_FIXED_STOP_WITH_MOVING_TO_TARGET_POSITION:
                                                                // Execute moving to target position
                                                                _instMoveAbsolute(Axis := _refPosAxis^,
                                                                                Execute := TRUE,
                                                                                Position := config.homing.extendedModeTargetPosition);

                                                                // Evaluate MC_Command
                                                                IF (_instMoveAbsolute.Done = TRUE) AND (_instTorqueLimiting.InClamping = FALSE) THEN
                                                                    // Homeposition reached - Set next state
                                                                    _exeOfBasicMotion := CMD_DONE;
                                                                    _homingSubState := HOMING_IDLE;

                                                                ELSIF (_instMoveAbsolute.Error = TRUE) THEN
                                                                    // Errorhandling
                                                                    _status := AxisStatus#ERR_MC_MOVEABSOLUTE;
                                                                    _statusText := STRING#'ERR_MC_MOVEABSOLUTE';
                                                                    _errorAutoCleared := TRUE;
                                                                    _diagnostics.subfunctionStatus := _instMoveAbsolute.ErrorId;
                                                                    _subfunctionStatus := _instMoveAbsolute.ErrorId;
                                                                    // Set next state
                                                                    _state := AXIS_STOP_ON_ERROR_SELECTION;
                                                                    _basicMotionState := CMD_BUSY;
                                                                    _activeHomingState := STANDARD_HOMING;
                                                                    _exeOfBasicMotion := CMD_ERROR;
                                                                    _homingSubState := HOMING_IDLE;

                                                                ELSIF (_instMoveAbsolute.CommandAborted = TRUE) THEN
                                                                    // Set next state
                                                                    _exeOfBasicMotion := CMD_ABORTED;
                                                                    _homingSubState := HOMING_IDLE;

                                                                // ELSE
                                                                    //   ; // Wait for reaching homeposition
                                                                END_IF;
                                                        END_CASE;
                                                ELSE
                                                    // Errorhandling
                                                    _status := AxisStatus#ERR_UNDEFINED_EXTENDED_HOMING_SUBSTATE;
                                                    _statusText := STRING#'ERR_UNDEFINED_EXTENDED_HOMING_SUBSTATE';
                                                    _errorUserCleared := TRUE;
                                                    _diagnostics.subfunctionStatus := WORD#0000;
                                                    _subfunctionStatus := AxisStatus#STATUS_NO_CALL;
                                                    // Set errorstate
                                                    _state := FB_ERROR;
                                                    tempStateChangeActive := FALSE;
                                                END_CASE;

                                            UNTIL (tempStateChangeActive = FALSE) // Repeat execution if a state is changing
                                            END_REPEAT;

                                        CMD_DONE,
                                        CMD_ABORTED,
                                        CMD_ERROR:
                                            // Return to NO_SELECTION if command finished
                                            IF (_basicCommand.%X10 = FALSE) // homing = FALSE
                                            THEN
                                                // Return to NO_HOMING_ACTIVE if command finished
                                                _basicMotionState := NO_SELECTION;
                                                _activeHomingState := STANDARD_HOMING;
                                                _exeOfBasicMotion := CMD_BUSY;
                                                _homingSubState := HOMING_IDLE;
                                            END_IF;
                                        ELSE
                                            // Errorhandling
                                            _status := AxisStatus#ERR_UNDEFINED_EXTENDED_HOMING_STATE;
                                            _statusText := STRING#'ERR_UNDEFINED_EXTENDED_HOMING_STATE';
                                            _errorUserCleared := TRUE;
                                            _diagnostics.subfunctionStatus := WORD#0000;
                                            _subfunctionStatus := AxisStatus#STATUS_NO_CALL;
                                            // Set errorstate
                                            _state := FB_ERROR;
                                    END_CASE;

                            ELSE
                                // Errorhandling
                                _status := AxisStatus#ERR_INVALID_HOMING_EXTENDED_MODE;
                                _statusText := STRING#'ERR_INVALID_HOMING_EXTENDED_MODE';
                                _errorAutoCleared := TRUE;
                                _diagnostics.subfunctionStatus := WORD#0000;
                                _subfunctionStatus := AxisStatus#STATUS_NO_CALL;
                                // Set next state
                                _state := AXIS_STOP_ON_ERROR_SELECTION;
                                _basicMotionState := NO_SELECTION;
                                _activeHomingState := STANDARD_HOMING;
                                _basicMotionState := NO_SELECTION;
                            END_CASE;

                        GEAR_IN_RELATIVE_SELECTED:
                            // Additional features (applicative): Change setpoint on the fly (gear ratio)

                            // Firstcycle of command
                            IF (_firstCycleBasicMotion = TRUE) THEN
                                // Reset GEAR_IN command
                                _instGearIn(Master := _refMasterAxis^,
                                            Slave := _refSyncAxis^,
                                            Execute := FALSE);

                                _instGearIn.RatioNumerator := config.gearInRelative.ratioNumerator;
                                _ratioNumerator := config.gearInRelative.ratioNumerator;
                                _instGearIn.RatioDenominator := config.gearInRelative.ratioDenominator;
                                _ratioDenominator := config.gearInRelative.ratioDenominator;
                                _instGearIn.Acceleration := config.gearInRelative.acceleration;
                                _basicAcceleration := config.gearInRelative.acceleration;
                                _instGearIn.Deceleration := config.gearInRelative.deceleration;
                                _basicDeceleration := config.gearInRelative.deceleration;
                                _instGearIn.Jerk := config.gearInRelative.jerk;
                                _basicJerk := config.gearInRelative.jerk;
                                _ratioChangeOnTheFly := config.gearInRelative.ratioChangeOnTheFly;

                            ELSIF ((_ratioChangeOnTheFly = TRUE) // Flying change of ratio numerator
                                AND ((config.gearInRelative.ratioNumerator <> _ratioNumerator)
                                OR (config.gearInRelative.ratioDenominator <> _ratioDenominator)))
                                AND
                                (_instGearIn.CommandAborted = FALSE)
                            THEN
                                _instGearIn(Master := _refMasterAxis^,
                                            Slave := _refSyncAxis^,
                                            Execute := FALSE);

                                _instGearIn.RatioNumerator := config.gearInRelative.ratioNumerator;
                                _ratioNumerator := config.gearInRelative.ratioNumerator;   // Apply the new gear ratio numerator
                                _instGearIn.RatioDenominator := config.gearInRelative.ratioDenominator;
                                _ratioDenominator := config.gearInRelative.ratioDenominator; // Apply the new gear ratio denominator

                                // Copy also dynamics
                                _instGearIn.Acceleration := config.gearInRelative.acceleration;
                                _basicAcceleration := config.gearInRelative.acceleration;
                                _instGearIn.Deceleration := config.gearInRelative.deceleration;
                                _basicDeceleration := config.gearInRelative.deceleration;
                                _instGearIn.Jerk := config.gearInRelative.jerk;
                                _basicJerk := config.gearInRelative.jerk;
                            END_IF;

                            // Call MC_Command
                            _instGearIn(Master := _refMasterAxis^,
                                        Slave := _refSyncAxis^,
                                        Execute := _basicCommand.%X7 OR _firstCycleBasicMotion); // Input: gearInRelative

                            // Evaluate MC_Command
                            IF (_instGearIn.Busy = FALSE) AND
                                (_instGearIn.Error = FALSE) AND
                                (_instGearIn.CommandAborted = FALSE) AND
                                (_instGearIn.InGear = FALSE)
                            THEN
                                // Return to NO_SELECTION if command finished
                                _basicMotionState := NO_SELECTION;

                            ELSIF (_instGearIn.Error = TRUE) THEN
                                // Errorhandling
                                _status := AxisStatus#ERR_MC_GEARIN;
                                _statusText := STRING#'ERR_MC_GEARIN';
                                _errorAutoCleared := TRUE;
                                _diagnostics.subfunctionStatus := _instGearIn.ErrorId;
                                _subfunctionStatus := _instGearIn.ErrorId;
                                _ratioChangeOnTheFly := FALSE;
                                // Set next state
                                _state := AXIS_STOP_ON_ERROR_SELECTION;
                                _basicMotionState := NO_SELECTION;
                            // ELSE
                                //   ; // Command selected
                            END_IF;

                            // Write MC_Command outputs to internal variable
                            _exeOfBasicMotion := 16#0;
                            _exeOfBasicMotion.%X0 := _instGearIn.Busy;
                            _exeOfBasicMotion.%X2 := _instGearIn.CommandAborted;
                            _exeOfBasicMotion.%X3 := _instGearIn.Error;
                            //#statExeOfBasicMotion.%X6 := tempStatusWord.%X21 AND NOT instGearIn.InGear; // write Synchronizing only when bit of instance of MC_GearIn.InGear = FALSE
                            _exeOfBasicMotion.%X7 := _instGearIn.InGear;

                        GEAR_IN_ABSOLUTE_SELECTED:
                            // Additional features (applicative): Change setpoint on the fly (gear ratio)

                            // Firstcycle of command
                            IF (_firstCycleBasicMotion = TRUE) THEN
                                // Reset GEAR_IN_POS command
                                _instGearInPos(Master := _refMasterAxis^,
                                               Slave := _refSyncAxis^,
                                               Execute := FALSE);

                                _instGearInPos.RatioNumerator := config.gearInAbsolute.ratioNumerator;
                                _ratioNumerator := config.gearInAbsolute.ratioNumerator;
                                _instGearInPos.RatioDenominator := config.gearInAbsolute.ratioDenominator;
                                _ratioDenominator := config.gearInAbsolute.ratioDenominator;

                                _instGearInPos.MasterSyncPosition := config.gearInAbsolute.masterSyncPosition;
                                _instGearInPos.SlaveSyncPosition := config.gearInAbsolute.slaveSyncPosition;
                                _instGearInPos.SyncProfileReference := config.gearInAbsolute.syncProfileReference;
                                _instGearInPos.MasterStartDistance := config.gearInAbsolute.masterStartDistance;
                                _instGearInPos.Velocity := config.gearInAbsolute.velocity;
                                _instGearInPos.Acceleration := config.gearInAbsolute.acceleration;
                                _instGearInPos.Deceleration := config.gearInAbsolute.deceleration;
                                _instGearInPos.Jerk := config.gearInAbsolute.jerk;
                                _instGearInPos.SyncDirection := config.gearInAbsolute.syncDirection;

                                _ratioChangeOnTheFly := config.gearInAbsolute.ratioChangeOnTheFly;

                            ELSIF (((_ratioChangeOnTheFly = TRUE) AND (config.gearInAbsolute.ratioNumerator <> _ratioNumerator))
                                OR ((_ratioChangeOnTheFly = TRUE) AND (config.gearInAbsolute.ratioDenominator <> _ratioDenominator)))
                                AND
                                (_instGearInPos.CommandAborted = FALSE)
                            THEN
                                _instGearInPos(Master := _refMasterAxis^,
                                            Slave := _refSyncAxis^,
                                            Execute := FALSE);

                                _instGearInPos.RatioNumerator := config.gearInAbsolute.ratioNumerator;
                                _ratioNumerator := config.gearInAbsolute.ratioNumerator;
                                _instGearInPos.RatioDenominator := config.gearInAbsolute.ratioDenominator;
                                _ratioDenominator := config.gearInAbsolute.ratioDenominator;

                                // Copy also dynamics
                                _instGearInPos.MasterSyncPosition := config.gearInAbsolute.masterSyncPosition;
                                _instGearInPos.SlaveSyncPosition := config.gearInAbsolute.slaveSyncPosition;
                                _instGearInPos.SyncProfileReference := config.gearInAbsolute.syncProfileReference;
                                _instGearInPos.MasterStartDistance := config.gearInAbsolute.masterStartDistance;
                                _instGearInPos.Velocity := config.gearInAbsolute.velocity;
                                _instGearInPos.Acceleration := config.gearInAbsolute.acceleration;
                                _instGearInPos.Deceleration := config.gearInAbsolute.deceleration;
                                _instGearInPos.Jerk := config.gearInAbsolute.jerk;
                                _instGearInPos.SyncDirection := config.gearInAbsolute.syncDirection;
                            END_IF;

                            // Call MC_Command
                            _instGearInPos(Master := _refMasterAxis^,
                                           Slave := _refSyncAxis^,
                                           Execute := _basicCommand.%X8 OR _firstCycleBasicMotion); // Input: gearInAbsolute

                            // Evaluate MC_Command
                            IF (_instGearInPos.Busy = FALSE) AND
                                (_instGearInPos.Error = FALSE) AND
                                (_instGearInPos.CommandAborted = FALSE) AND
                                (_instGearInPos.StartSync = FALSE) AND
                                (_instGearInPos.InSync = FALSE)
                            THEN
                                // Return to NO_SELECTION if command finished
                                _basicMotionState := NO_SELECTION;

                            ELSIF (_instGearInPos.Error = TRUE) THEN
                                // Errorhandling
                                _status := AxisStatus#ERR_MC_GEARINPOS;
                                _statusText := STRING#'ERR_MC_GEARINPOS';
                                _errorAutoCleared := TRUE;
                                _diagnostics.subfunctionStatus := _instGearInPos.ErrorId;
                                _subfunctionStatus := _instGearInPos.ErrorId;
                                _ratioChangeOnTheFly := FALSE;
                                // Set next state
                                _state := AXIS_STOP_ON_ERROR_SELECTION;
                                _basicMotionState := NO_SELECTION;
                            // ELSE
                                //   ; // Command selected
                            END_IF;

                            // Write MC_Command outputs to internal variable
                            _exeOfBasicMotion := 16#0;
                            _exeOfBasicMotion.%X0 := _instGearInPos.Busy;
                            _exeOfBasicMotion.%X2 := _instGearInPos.CommandAborted;
                            _exeOfBasicMotion.%X3 := _instGearInPos.Error;
                            _exeOfBasicMotion.%X6 := _instGearInPos.StartSync;
                            _exeOfBasicMotion.%X7 := _instGearInPos.InSync;

                        GEAR_IN_VELOCITY_SELECTED:

                            // Firstcycle of command
                            IF (_firstCycleBasicMotion = TRUE) THEN
                                // Reset GEAR_IN_VELOCITY command
                                _instGearInVelocity(Master := _refMasterAxis^,
                                                    Slave := _refSyncAxis^,
                                                    Execute := FALSE,
                                                    Acceleration := config.gearInVelocity.acceleration,
                                                    Deceleration := config.gearInVelocity.deceleration,
                                                    Jerk := config.gearInVelocity.jerk,
                                                    PositionControlled := config.gearInVelocity.positionControlled);
                            END_IF;

                            // Call MC_Command
                            _instGearInVelocity(Master := _refMasterAxis^,
                                                Slave := _refSyncAxis^,
                                                Execute := _basicCommand.%X12 OR _firstCycleBasicMotion, // Input: gearInVelocity
                                                ContinuousUpdate := config.gearInVelocity.continuousUpdate,
                                                RatioNumerator := config.gearInVelocity.ratioNumerator,
                                                RatioDenominator := config.gearInVelocity.ratioDenominator);

                            // Evaluate MC_Command
                            IF (_instGearInVelocity.Busy = FALSE) AND
                                (_instGearInVelocity.Error = FALSE) AND
                                (_instGearInVelocity.CommandAborted = FALSE) AND
                                (_instGearInVelocity.StartSync = FALSE) AND
                                (_instGearInVelocity.InSync = FALSE)
                            THEN
                                // Return to NO_SELECTION if command finished
                                _basicMotionState := NO_SELECTION;

                            ELSIF (_instGearInVelocity.Error = TRUE) THEN
                                // Errorhandling
                                _status := AxisStatus#ERR_MC_GEARINVELOCITY;
                                _statusText := STRING#'ERR_MC_GEARINVELOCITY';
                                _errorAutoCleared := TRUE;
                                _diagnostics.subfunctionStatus := _instGearInVelocity.ErrorId;
                                _subfunctionStatus := _instGearInVelocity.ErrorId;
                                // Set next state
                                _state := AXIS_STOP_ON_ERROR_SELECTION;
                                _basicMotionState := NO_SELECTION;
                            // ELSE
                            //   ; // Command selected
                            END_IF;

                            // Write MC_Command outputs to internal variable
                            _exeOfBasicMotion := 16#0;
                            _exeOfBasicMotion.%X0 := _instGearInVelocity.Busy;
                            _exeOfBasicMotion.%X2 := _instGearInVelocity.CommandAborted;
                            _exeOfBasicMotion.%X3 := _instGearInVelocity.Error;
                            _exeOfBasicMotion.%X6 := _instGearInVelocity.StartSync;
                            _exeOfBasicMotion.%X7 := _instGearInVelocity.InSync;

                        CAM_IN_SELECTED:

                            // Firstcycle of command
                            IF (_firstCycleBasicMotion = TRUE) THEN
                                // Reset CAM_IN command
                                _instCamIn(Master := _refMasterAxis^,
                                           Slave := _refSyncAxis^,
                                           Cam := _refCamBase^,
                                           Execute := FALSE,
                                           MasterOffset := config.camIn.masterOffset,
                                           SlaveOffset := config.camIn.slaveOffset,
                                           MasterScaling := config.camIn.masterScaling,
                                           SlaveScaling := config.camIn.slaveScaling,
                                           MasterSyncPosition := config.camIn.masterSyncPosition,
                                           SyncProfileReference := config.camIn.syncProfileReference,
                                           MasterStartDistance := config.camIn.masterStartDistance,
                                           Velocity := config.camIn.velocity,
                                           Acceleration := config.camIn.acceleration,
                                           Deceleration := config.camIn.deceleration,
                                           Jerk := config.camIn.jerk,
                                           ApplicationMode := config.camIn.applicationMode,
                                           SyncDirection := config.camIn.syncDirection);

                                _applicationMode := config.camIn.applicationMode;
                            END_IF;

                            // Call MC_Command
                            _instCamIn(Master := _refMasterAxis^,
                                       Slave := _refSyncAxis^,
                                       Cam := _refCamBase^,
                                       Execute := _basicCommand.%X9 OR _firstCycleBasicMotion); // Input: camIn

                            // Evaluate MC_Command
                            IF ((_instCamIn.Busy = FALSE) AND
                                (_instCamIn.Error = FALSE) AND
                                (_instCamIn.CommandAborted = FALSE) AND
                                (_instCamIn.InSync = FALSE) AND
                                (_instCamIn.StartSync = FALSE) AND
                                (_basicCommand.%X9 = FALSE))
                                AND // Wait for one cycle EndOfProfile (--> Done) before function is finished at applicationMode ONCE
                                ((_applicationMode <> APPLICATION_MODE_ONCE) OR
                                ((_applicationMode = APPLICATION_MODE_ONCE) AND (_instCamIn.EndOfProfile = FALSE)))
                            THEN
                                // Return to NO_SELECTION if command finished
                                _basicMotionState := NO_SELECTION;
